{attribute 'linkalways'} 
{attribute 'no_explicit_call' := 'This FB is a CLASS and must be accessed using methods or properties'}
{attribute 'enable_dynamic_creation'}
FUNCTION_BLOCK _ETcVnSta EXTENDS EnumDatatypeBase
VAR
	localData : ETcVnSta;
	activeData : REFERENCE TO ETcVnSta;
	enumBaseDatatype : _UDINT(localData);
END_VAR

METHOD PRIVATE AddLocalEnumeration
VAR_INPUT
	Enumeration : T_MAXSTRING;
	Value : ETcVnSta;
END_VAR
AddEnumeration(Enumeration, Value);
END_METHOD

PROPERTY PUBLIC Address : PVOID
GET
Address := ADR(activeData);
END_GET
END_PROPERTY

METHOD PUBLIC ClearReference
VAR_INPUT
END_VAR
activeData REF= localData;
SetBaseDatatypeReference();
END_METHOD

METHOD PUBLIC Clone : I_Datatype
VAR
    pClone : POINTER TO _ETcVnSta;
END_VAR
pClone := __NEW(_ETcVnSta(InitialValue := Value));
Clone := pClone^;
END_METHOD

METHOD FB_init : BOOL
VAR_INPUT
	bInitRetains : BOOL; // if TRUE, the retain variables are initialized (warm start / cold start)
	bInCopyCode : BOOL;  // if TRUE, the instance afterwards gets moved into the copy code (online change)
	InitialValue : ETcVnSta;
END_VAR
localData := InitialValue;
AddBaseDatatype(enumBaseDatatype);
ClearReference();

AddLocalEnumeration('TCVN_STA_CLASSIFIER', ETcVnSta.TCVN_STA_CLASSIFIER);
AddLocalEnumeration('TCVN_STA_NOVELTY_DETECTOR', ETcVnSta.TCVN_STA_NOVELTY_DETECTOR);
AddLocalEnumeration('TCVN_STA_REGRESSOR', ETcVnSta.TCVN_STA_REGRESSOR);
AddLocalEnumeration('TCVN_STA_CLUSTERER', ETcVnSta.TCVN_STA_CLUSTERER);
END_METHOD

PROPERTY PUBLIC Identifier : T_MAXSTRING
GET
Identifier := 'ETcVnSta';
END_GET
END_PROPERTY

METHOD IsEnumeratorValueEqual : BOOL
VAR_INPUT
	Enumerator : I_KeyValueForwardEnumerator;
END_VAR
VAR
	storedValue : ETcVnSta;
END_VAR
IF NOT Enumerator.TryGet(storedValue) THEN
	RETURN;
END_IF

IsEnumeratorValueEqual := storedValue = activeData;
END_METHOD

METHOD PUBLIC MakeReferenceTo
VAR_INPUT
	ReferenceTarget : REFERENCE TO ETcVnSta;
END_VAR
activeData REF= ReferenceTarget;
SetBaseDatatypeReference();
END_METHOD

METHOD PROTECTED SetBaseDatatypeReference
VAR_INPUT
END_VAR
enumBaseDatatype.MakeReferenceTo(activeData);
END_METHOD

PROPERTY PUBLIC Size : UDINT
GET
Size := SIZEOF(activeData);
END_GET
END_PROPERTY

METHOD TryMakeReferenceTo : BOOL
VAR_INPUT
	Target : I_Datatype;
END_VAR
VAR
	targetAsEnum : I_EnumDatatype;
	pTargetData : POINTER TO ETcVnSta;
END_VAR
IF NOT Target.TryResolveAsEnumDatatype(targetAsEnum) THEN
	RETURN;
END_IF

IF targetAsEnum.Identifier <> Identifier THEN
	RETURN;
END_IF

pTargetData := Target.Address;
activeData REF= pTargetData^;
SetBaseDatatypeReference();
TryMakeReferenceTo := TRUE;
END_METHOD

PROPERTY PUBLIC Value : ETcVnSta
GET
Value := activeData;
END_GET
SET
activeData := Value;
END_SET
END_PROPERTY

END_FUNCTION_BLOCK

(* stored: Version 1.1.0.1
   POU _ETcVnSta: Id {7dd43c9d-8ac3-4e90-9e41-ec146f363131}, SpecialFunc None
   Folder Constructor: Id {c1f03731-4168-4362-a278-8879773f5ce3}
   Folder Private: Id {29c7ae29-4473-4539-bebc-557670e0a6ee}
   Folder Protected: Id {62b7b728-94a9-4018-84a7-4e1171a0aa2d}
   Method AddLocalEnumeration: Id {47dd97d4-4817-4cce-98a1-d2d754bf3c11}
   Property Address: Id {26052fc0-5926-47c8-a519-9487114b2358}
   Get Get: Id {51d93502-7123-4bb9-a564-16b60f119bbc}
   Method ClearReference: Id {ff03292f-9b97-4f9f-9fe2-f92f29bcf430}
   Method Clone: Id {beac26d5-897e-4fb9-ac90-7d9391d8c741}
   Method FB_init: Id {4fd2d8e8-5d20-42b9-95f9-52b2c6c65f09}
   Property Identifier: Id {f543bada-c7b4-4913-86e3-5f19a72c61ec}
   Get Get: Id {af88c44c-9b5e-4138-89a0-8fe2d7addab3}
   Method IsEnumeratorValueEqual: Id {259c3cf6-e6ab-4e43-8b5c-64eee7770457}
   Method MakeReferenceTo: Id {3c027c9a-2383-4ea9-be6a-1c23fbc69ade}
   Method SetBaseDatatypeReference: Id {9204a2a0-f156-483e-9460-3739df787e42}
   Property Size: Id {658617aa-d31e-44b3-98f8-bcab1be385bf}
   Get Get: Id {125da7bc-8209-4d7e-9051-919fd586c52e}
   Method TryMakeReferenceTo: Id {fce58ce8-ec4b-412d-be9c-3592aaa82bd3}
   Property Value: Id {3bb5b0dc-f6dc-4648-ab0c-ee4e30a1d1b0}
   Get Get: Id {c0ca85d0-6ee8-478f-854d-7836c5ce37e8}
   Set Set: Id {6a4ea26d-967a-449f-8081-4af6ac1d1c4a} *)
